KUKA KRL program: ps_p13060r5_all_resp_x1.src, ps_p13060r5_all_resp_x1.dat

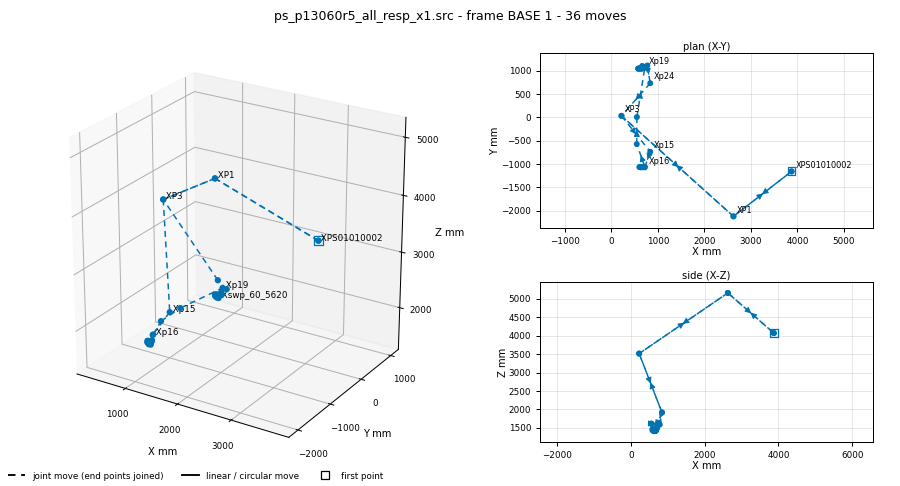
[picture p0: tool path of ps_p13060r5_all_resp_x1.src in frame BASE 1, 36 of 36 moves have a stored position in this frame; points joined in program order, loops and branches not executed]
--- ps_p13060r5_all_resp_x1.src ---
&ACCESS RVO1
&REL 27
&COMMENT SOLDA ACTROS GUN X1
&PARAM DISKPATH = KRC:\R1\Program
DEF ps_p13060r5_all_resp_x1( )
;FOLD INI
  ;FOLD BASISTECH INI
    GLOBAL INTERRUPT DECL 3 WHEN $STOPMESS==TRUE DO IR_STOPM ( )
    INTERRUPT ON 3
    BAS (#INITMOV,0 )
  ;ENDFOLD (BASISTECH INI)
;FOLD SPOTTECH INI
USERSPOT(#INIT)
;ENDFOLD (SPOTTECH INI)
;FOLD GRIPPERTECH INI

;ENDFOLD (GRIPPERTECH INI)
  ;FOLD USER INI
    ;Make your modifications here

     ;FOLD COLLISION_V_3.01 INI ;%{E}
        IF (COLLISION_DATA[1].I_NR>0) THEN
          GLOBAL INTERRUPT DECL 21 WHEN $IN[COLLISION_DATA[1].I_NR]==FALSE DO COLLSTOP (1,0 )
        ENDIF
        IF (COLLISION_DATA[2].I_NR>0) THEN
          GLOBAL INTERRUPT DECL 22 WHEN $IN[COLLISION_DATA[2].I_NR]==FALSE DO COLLSTOP (2,0 )
        ENDIF
        IF (COLLISION_DATA[3].I_NR>0) THEN
          GLOBAL INTERRUPT DECL 23 WHEN $IN[COLLISION_DATA[3].I_NR]==FALSE DO COLLSTOP (3,0 )
        ENDIF
        IF (COLLISION_DATA[4].I_NR>0) THEN
          GLOBAL INTERRUPT DECL 24 WHEN $IN[COLLISION_DATA[4].I_NR]==FALSE DO COLLSTOP (4,0 )
        ENDIF
     ;ENDFOLD (Collision)

  ;ENDFOLD (USER INI)
;ENDFOLD (INI)

; Caracterização dos meios de produção: P13.060-R5
; Versão atual: 17/07/2013 Nome: Solda Respot X1
; Change: LTA/LTA/MGS/MHSB/STB

chk_w1_wechs_ok ( )           ; VERIFICAÇÃO DE FERRAMENA: X1

;FOLD PTP PS01010002 Vel=100 % PDAT23 Tool[1]:Gun X1 Base[1]:Actros;%{PE}%R 8.2.20,%MKUKATPBASIS,%CMOVE,%VPTP,%P 1:PTP, 2:PS01010002, 3:, 5:100, 7:PDAT23
$BWDSTART=FALSE
PDAT_ACT=PPDAT23
FDAT_ACT=FPS01010002
BAS(#PTP_PARAMS,100)
PTP XPS01010002
;ENDFOLD

IF MaxStandMenge (3) THEN
 MaxStandmengeErreicht (3)
ENDIF

IF Elektrodenwechsel (3) THEN
 e_Fraes_1 ()
ENDIF


;FOLD PTP P1 CONT Vel=100 % PDAT15 Tool[1]:Gun X1 Base[1]:Actros;%{PE}%R 8.2.20,%MKUKATPBASIS,%CMOVE,%VPTP,%P 1:PTP, 2:P1, 3:C_DIS, 5:100, 7:PDAT15
$BWDSTART=FALSE
PDAT_ACT=PPDAT15
FDAT_ACT=FP1
BAS(#PTP_PARAMS,100)
PTP XP1 C_DIS
;ENDFOLD
;FOLD PTP P3 CONT Vel=100 % PDAT18 Tool[1]:Gun X1 Base[1]:Actros;%{PE}%R 8.2.20,%MKUKATPBASIS,%CMOVE,%VPTP,%P 1:PTP, 2:P3, 3:C_DIS, 5:100, 7:PDAT18
$BWDSTART=FALSE
PDAT_ACT=PPDAT18
FDAT_ACT=FP3
BAS(#PTP_PARAMS,100)
PTP XP3 C_DIS
;ENDFOLD
;FOLD PTP p15 CONT Vel=100 % P_OLP2 Tool[1]:Gun X1 Base[1]:Actros;%{PE}%R 8.2.20,%MKUKATPBASIS,%CMOVE,%VPTP,%P 1:PTP, 2:p15, 3:C_DIS, 5:100, 7:P_OLP2
$BWDSTART=FALSE
PDAT_ACT=PP_OLP2
FDAT_ACT=Fp15
BAS(#PTP_PARAMS,100)
PTP Xp15 C_DIS
;ENDFOLD

;FOLD Collision.Monitoring_1_On ;%{PE}%MKUKATPUSER
COLLSTOP( 1, 1 ) ;Interrupt-Controlled
;ENDFOLD

;FOLD OUT 3339 'R5 SOLDANDO' State=TRUE ;%{PE}%R 8.2.20,%MKUKATPBASIS,%COUT,%VOUTX,%P 2:3339, 3:R5 SOLDANDO, 5:TRUE, 6:
$OUT[3339]=TRUE
;ENDFOLD
;FOLD OUT 3340 'locking-signal PLC' State=FALSE ;%{PE}%R 8.2.20,%MKUKATPBASIS,%COUT,%VOUTX,%P 2:3340, 3:locking-signal PLC, 5:FALSE, 6:
$OUT[3340]=FALSE
;ENDFOLD

;FOLD PTP p16 CONT Vel=100 % P_OLP3 Tool[1]:Gun X1 Base[1]:Actros;%{PE}%R8.2,%MKUKATPBASIS,%CMOVE,%VPTP,%P 1:PTP, 2:p16, 3:C_DIS, 5:100, 7:P_OLP3
$BWDSTART = FALSE
PDAT_ACT= PP_OLP3
FDAT_ACT= Fp16
BAS(#PTP_PARAMS,100)
PTP Xp16 C_DIS
;ENDFOLD
;FOLD PTP P7 CONT Vel=100 % PDAT22 Tool[1]:Gun X1 Base[1]:Actros;%{PE}%R 8.2.20,%MKUKATPBASIS,%CMOVE,%VPTP,%P 1:PTP, 2:P7, 3:C_DIS, 5:100, 7:PDAT22
$BWDSTART=FALSE
PDAT_ACT=PPDAT22
FDAT_ACT=FP7
BAS(#PTP_PARAMS,100)
PTP XP7 C_DIS
;ENDFOLD
;FOLD PTP p17 PDAT1 RETR CLS Gun=3 Tool[1]:Gun X1 Base[1]:Actros;%{PE}%R 8.2.2,%MKUKATPSPOT,%CRETR,%VPTP,%P 1:PTP, 2:p17, 3:, 5:100, 7:PDAT1, 9:#CLO, 11:3, 13:#FIRST
$BWDSTART=FALSE
PDAT_ACT=PPDAT1
FDAT_ACT=Fp17
BAS(#PTP_PARAMS,PPDAT1.VEL)
S_ACT.GUN=3
S_ACT.PAIR=#FIRST
S_ACT.RETR=#CLO
S_READY=FALSE
PTP Xp17
USERSPOT(#RETR, S_ACT)
WAIT FOR S_READY
;ENDFOLD

;FOLD ; SWP_60_5617;%{PE}%R 8.2.20,%MKUKATPBASIS,%CCOMMENT,%VNORMAL,%P 2:SWP_60_5617
;ENDFOLD
;FOLD PTP swp_60_5617 PDAT2 SPOT Gun=3 RETR CLS PGNO1=121 ACTIVE=1 Tool[1]:Gun X1 Base[1]:Actros;%{PE}%R 8.2.2,%MKUKATPSPOT,%CSPOT,%VPTP,%P 1:PTP, 2:swp_60_5617, 3:, 5:100, 7:PDAT2, 10:3, 12:#FIRST, 14:#CLO, 16:171, 18:1, 20:0, 22:0, 24:1, 25:NORMAL
$BWDSTART=FALSE
PDAT_ACT=PPDAT2
FDAT_ACT=Fswp_60_5617
BAS(#PTP_PARAMS,PPDAT2.VEL)
S_ACT.GUN=3
S_ACT.PAIR=SDEFAULT.PAIR
S_ACT.RETR=#CLO
S_ACT.CLO_TM=1
S_ACT.PGNO1=121
S_ACT.PGNO2=SDEFAULT.PGNO2
S_ACT.PRESS1=SDEFAULT.PRESS1
S_ACT.PRESS2=SDEFAULT.PRESS2
S_READY=FALSE
PTP Xswp_60_5617
USERSPOT(#SPOT, S_ACT)
WAIT FOR S_READY
;ENDFOLD

;FOLD ; SWP_60_5619;%{PE}%R 8.2.20,%MKUKATPBASIS,%CCOMMENT,%VNORMAL,%P 2:SWP_60_5619
;ENDFOLD
;FOLD PTP swp_60_5619 PDAT3 SPOT Gun=3 RETR CLS PGNO1=122 ACTIVE=1 Tool[1]:Gun X1 Base[1]:Actros;%{PE}%R 8.2.2,%MKUKATPSPOT,%CSPOT,%VPTP,%P 1:PTP, 2:swp_60_5619, 3:, 5:100, 7:PDAT3, 10:3, 12:#FIRST, 14:#CLO, 16:172, 18:1, 20:0, 22:0, 24:1, 25:NORMAL
$BWDSTART=FALSE
PDAT_ACT=PPDAT3
FDAT_ACT=Fswp_60_5619
BAS(#PTP_PARAMS,PPDAT3.VEL)
S_ACT.GUN=3
S_ACT.PAIR=SDEFAULT.PAIR
S_ACT.RETR=#CLO
S_ACT.CLO_TM=1
S_ACT.PGNO1=122
S_ACT.PGNO2=SDEFAULT.PGNO2
S_ACT.PRESS1=SDEFAULT.PRESS1
S_ACT.PRESS2=SDEFAULT.PRESS2
S_READY=FALSE
PTP Xswp_60_5619
USERSPOT(#SPOT, S_ACT)
WAIT FOR S_READY
;ENDFOLD

;FOLD ; SWP_60_5615;%{PE}%R 8.2.20,%MKUKATPBASIS,%CCOMMENT,%VNORMAL,%P 2:SWP_60_5615
;ENDFOLD
;FOLD PTP swp_60_5615 PDAT4 SPOT Gun=3 RETR CLS PGNO1=123 ACTIVE=1 Tool[1]:Gun X1 Base[1]:Actros;%{PE}%R 8.2.2,%MKUKATPSPOT,%CSPOT,%VPTP,%P 1:PTP, 2:swp_60_5615, 3:, 5:100, 7:PDAT4, 10:3, 12:#FIRST, 14:#CLO, 16:173, 18:1, 20:0, 22:0, 24:1, 25:NORMAL
$BWDSTART=FALSE
PDAT_ACT=PPDAT4
FDAT_ACT=Fswp_60_5615
BAS(#PTP_PARAMS,PPDAT4.VEL)
S_ACT.GUN=3
S_ACT.PAIR=SDEFAULT.PAIR
S_ACT.RETR=#CLO
S_ACT.CLO_TM=1
S_ACT.PGNO1=123
S_ACT.PGNO2=SDEFAULT.PGNO2
S_ACT.PRESS1=SDEFAULT.PRESS1
S_ACT.PRESS2=SDEFAULT.PRESS2
S_READY=FALSE
PTP Xswp_60_5615
USERSPOT(#SPOT, S_ACT)
WAIT FOR S_READY
;ENDFOLD

;FOLD ; SWP_60_5613;%{PE}%R 8.2.20,%MKUKATPBASIS,%CCOMMENT,%VNORMAL,%P 2:SWP_60_5613
;ENDFOLD
;FOLD PTP swp_60_5613 PDAT5 SPOT Gun=3 RETR CLS PGNO1=124 ACTIVE=1 Tool[1]:Gun X1 Base[1]:Actros;%{PE}%R 8.2.2,%MKUKATPSPOT,%CSPOT,%VPTP,%P 1:PTP, 2:swp_60_5613, 3:, 5:100, 7:PDAT5, 10:3, 12:#FIRST, 14:#CLO, 16:174, 18:1, 20:0, 22:0, 24:1, 25:NORMAL
$BWDSTART=FALSE
PDAT_ACT=PPDAT5
FDAT_ACT=Fswp_60_5613
BAS(#PTP_PARAMS,PPDAT5.VEL)
S_ACT.GUN=3
S_ACT.PAIR=SDEFAULT.PAIR
S_ACT.RETR=#CLO
S_ACT.CLO_TM=1
S_ACT.PGNO1=124
S_ACT.PGNO2=SDEFAULT.PGNO2
S_ACT.PRESS1=SDEFAULT.PRESS1
S_ACT.PRESS2=SDEFAULT.PRESS2
S_READY=FALSE
PTP Xswp_60_5613
USERSPOT(#SPOT, S_ACT)
WAIT FOR S_READY
;ENDFOLD

;FOLD LIN P8 CONT Vel=1 m/s CPDAT3 Tool[1]:Gun X1 Base[1]:Actros;%{PE}%R 8.2.20,%MKUKATPBASIS,%CMOVE,%VLIN,%P 1:LIN, 2:P8, 3:C_DIS C_DIS, 5:1, 7:CPDAT3
$BWDSTART=FALSE
LDAT_ACT=LCPDAT3
FDAT_ACT=FP8
BAS(#CP_PARAMS,1)
LIN XP8 C_DIS C_DIS
;ENDFOLD

;FOLD ; SWP_60_5611;%{PE}%R 8.2.20,%MKUKATPBASIS,%CCOMMENT,%VNORMAL,%P 2:SWP_60_5611
;ENDFOLD
;FOLD PTP swp_60_5611 PDAT6 SPOT Gun=3 RETR CLS PGNO1=125 ACTIVE=1 Tool[1]:Gun X1 Base[1]:Actros;%{PE}%R 8.2.2,%MKUKATPSPOT,%CSPOT,%VPTP,%P 1:PTP, 2:swp_60_5611, 3:, 5:100, 7:PDAT6, 10:3, 12:#FIRST, 14:#CLO, 16:175, 18:1, 20:0, 22:0, 24:1, 25:NORMAL
$BWDSTART=FALSE
PDAT_ACT=PPDAT6
FDAT_ACT=Fswp_60_5611
BAS(#PTP_PARAMS,PPDAT6.VEL)
S_ACT.GUN=3
S_ACT.PAIR=SDEFAULT.PAIR
S_ACT.RETR=#CLO
S_ACT.CLO_TM=1
S_ACT.PGNO1=125
S_ACT.PGNO2=SDEFAULT.PGNO2
S_ACT.PRESS1=SDEFAULT.PRESS1
S_ACT.PRESS2=SDEFAULT.PRESS2
S_READY=FALSE
PTP Xswp_60_5611
USERSPOT(#SPOT, S_ACT)
WAIT FOR S_READY
;ENDFOLD

;FOLD ; SWP_60_5605;%{PE}%R 8.2.20,%MKUKATPBASIS,%CCOMMENT,%VNORMAL,%P 2:SWP_60_5605
;ENDFOLD
;FOLD LIN swp_60_5605 CPDAT1 SPOT Gun=3 RETR CLS PGNO1=126 ACTIVE=1 Tool[1]:Gun X1 Base[1]:Actros;%{PE}%R 8.2.2,%MKUKATPSPOT,%CSPOT,%VLIN,%P 1:LIN, 2:swp_60_5605, 3:, 5:2, 7:CPDAT1, 10:3, 12:#FIRST, 14:#CLO, 16:176, 18:1, 20:0, 22:0, 24:1, 25:NORMAL
$BWDSTART=FALSE
LDAT_ACT=LCPDAT1
FDAT_ACT=Fswp_60_5605
BAS(#CP_PARAMS,LCPDAT1.VEL)
S_ACT.GUN=3
S_ACT.PAIR=SDEFAULT.PAIR
S_ACT.RETR=#CLO
S_ACT.CLO_TM=1
S_ACT.PGNO1=126
S_ACT.PGNO2=SDEFAULT.PGNO2
S_ACT.PRESS1=SDEFAULT.PRESS1
S_ACT.PRESS2=SDEFAULT.PRESS2
S_READY=FALSE
LIN Xswp_60_5605
USERSPOT(#SPOT, S_ACT)
WAIT FOR S_READY
;ENDFOLD

;FOLD ; SWP_60_5607;%{PE}%R 8.2.20,%MKUKATPBASIS,%CCOMMENT,%VNORMAL,%P 2:SWP_60_5607
;ENDFOLD
;FOLD LIN swp_60_5607 CPDAT4 SPOT Gun=3 RETR CLS PGNO1=127 ACTIVE=1 Tool[1]:Gun X1 Base[1]:Actros;%{PE}%R 8.2.2,%MKUKATPSPOT,%CSPOT,%VLIN,%P 1:LIN, 2:swp_60_5607, 3:, 5:2, 7:CPDAT4, 10:3, 12:#FIRST, 14:#CLO, 16:177, 18:1, 20:0, 22:0, 24:1, 25:NORMAL
$BWDSTART=FALSE
LDAT_ACT=LCPDAT4
FDAT_ACT=Fswp_60_5607
BAS(#CP_PARAMS,LCPDAT4.VEL)
S_ACT.GUN=3
S_ACT.PAIR=SDEFAULT.PAIR
S_ACT.RETR=#CLO
S_ACT.CLO_TM=1
S_ACT.PGNO1=127
S_ACT.PGNO2=SDEFAULT.PGNO2
S_ACT.PRESS1=SDEFAULT.PRESS1
S_ACT.PRESS2=SDEFAULT.PRESS2
S_READY=FALSE
LIN Xswp_60_5607
USERSPOT(#SPOT, S_ACT)
WAIT FOR S_READY
;ENDFOLD

;FOLD ; SWP_60_5609;%{PE}%R 8.2.20,%MKUKATPBASIS,%CCOMMENT,%VNORMAL,%P 2:SWP_60_5609
;ENDFOLD
;FOLD PTP swp_60_5609 PDAT9 SPOT Gun=3 RETR OPN PGNO1=128 ACTIVE=1 Tool[1]:Gun X1 Base[1]:Actros;%{PE}%R 8.2.2,%MKUKATPSPOT,%CSPOT,%VPTP,%P 1:PTP, 2:swp_60_5609, 3:, 5:100, 7:PDAT9, 10:3, 12:#FIRST, 14:#OPN, 16:178, 18:1, 20:0, 22:0, 24:1, 25:NORMAL
$BWDSTART=FALSE
PDAT_ACT=PPDAT9
FDAT_ACT=Fswp_60_5609
BAS(#PTP_PARAMS,PPDAT9.VEL)
S_ACT.GUN=3
S_ACT.PAIR=SDEFAULT.PAIR
S_ACT.RETR=#OPN
S_ACT.CLO_TM=1
S_ACT.PGNO1=128
S_ACT.PGNO2=SDEFAULT.PGNO2
S_ACT.PRESS1=SDEFAULT.PRESS1
S_ACT.PRESS2=SDEFAULT.PRESS2
S_READY=FALSE
PTP Xswp_60_5609
USERSPOT(#SPOT, S_ACT)
WAIT FOR S_READY
;ENDFOLD

;FOLD PTP p18 CONT Vel=100 % P_OLP13 Tool[1]:Gun X1 Base[1]:Actros;%{PE}%R8.2,%MKUKATPBASIS,%CMOVE,%VPTP,%P 1:PTP, 2:p18, 3:C_DIS, 5:100, 7:P_OLP13
$BWDSTART = FALSE
PDAT_ACT= PP_OLP13
FDAT_ACT= Fp18
BAS(#PTP_PARAMS,100)
PTP Xp18 C_DIS
;ENDFOLD
;FOLD PTP P6 CONT Vel=100 % PDAT21 Tool[1]:Gun X1 Base[1]:Actros;%{PE}%R 8.2.20,%MKUKATPBASIS,%CMOVE,%VPTP,%P 1:PTP, 2:P6, 3:C_DIS, 5:100, 7:PDAT21
$BWDSTART=FALSE
PDAT_ACT=PPDAT21
FDAT_ACT=FP6
BAS(#PTP_PARAMS,100)
PTP XP6 C_DIS
;ENDFOLD

;FOLD Collision.Monitoring_1_Off . ;%{PE}%MKUKATPUSER
COLLSTOP( 1, 2+0 )
;ENDFOLD
;FOLD Collision.Monitoring_2_On ;%{PE}%MKUKATPUSER
COLLSTOP( 2, 1 ) ;Interrupt-Controlled
;ENDFOLD

;FOLD PTP p26 CONT Vel=100 % PDAT10 Tool[1]:Gun X1 Base[1]:Actros;%{PE}%R 8.2.20,%MKUKATPBASIS,%CMOVE,%VPTP,%P 1:PTP, 2:p26, 3:C_DIS, 5:100, 7:PDAT10
$BWDSTART=FALSE
PDAT_ACT=PPDAT10
FDAT_ACT=Fp26
BAS(#PTP_PARAMS,100)
PTP Xp26 C_DIS
;ENDFOLD
;FOLD PTP p19 CONT Vel=100 % P_OLP14 Tool[1]:Gun X1 Base[1]:Actros;%{PE}%R8.2,%MKUKATPBASIS,%CMOVE,%VPTP,%P 1:PTP, 2:p19, 3:C_DIS, 5:100, 7:P_OLP14
$BWDSTART = FALSE
PDAT_ACT= PP_OLP14
FDAT_ACT= Fp19
BAS(#PTP_PARAMS,100)
PTP Xp19 C_DIS
;ENDFOLD
;FOLD PTP p20 CONT Vel=100 % PDAT12 Tool[1]:Gun X1 Base[1]:Actros;%{PE}%R 8.2.20,%MKUKATPBASIS,%CMOVE,%VPTP,%P 1:PTP, 2:p20, 3:C_DIS, 5:100, 7:PDAT12
$BWDSTART=FALSE
PDAT_ACT=PPDAT12
FDAT_ACT=Fp20
BAS(#PTP_PARAMS,100)
PTP Xp20 C_DIS
;ENDFOLD

;FOLD ; SWP_60_5610;%{PE}%R 8.2.20,%MKUKATPBASIS,%CCOMMENT,%VNORMAL,%P 2:SWP_60_5610
;ENDFOLD
;FOLD PTP swp_60_5610 PDAT13 SPOT Gun=3 RETR CLS PGNO1=129 ACTIVE=1 Tool[1]:Gun X1 Base[1]:Actros;%{PE}%R 8.2.2,%MKUKATPSPOT,%CSPOT,%VPTP,%P 1:PTP, 2:swp_60_5610, 3:, 5:100, 7:PDAT13, 10:3, 12:#FIRST, 14:#CLO, 16:179, 18:1, 20:0, 22:0, 24:1, 25:NORMAL
$BWDSTART=FALSE
PDAT_ACT=PPDAT13
FDAT_ACT=Fswp_60_5610
BAS(#PTP_PARAMS,PPDAT13.VEL)
S_ACT.GUN=3
S_ACT.PAIR=SDEFAULT.PAIR
S_ACT.RETR=#CLO
S_ACT.CLO_TM=1
S_ACT.PGNO1=129
S_ACT.PGNO2=SDEFAULT.PGNO2
S_ACT.PRESS1=SDEFAULT.PRESS1
S_ACT.PRESS2=SDEFAULT.PRESS2
S_READY=FALSE
PTP Xswp_60_5610
USERSPOT(#SPOT, S_ACT)
WAIT FOR S_READY
;ENDFOLD

;FOLD ; SWP_60_5608;%{PE}%R 8.2.20,%MKUKATPBASIS,%CCOMMENT,%VNORMAL,%P 2:SWP_60_5608
;ENDFOLD
;FOLD PTP swp_60_5608 PDAT14 SPOT Gun=3 RETR CLS PGNO1=130 ACTIVE=1 Tool[1]:Gun X1 Base[1]:Actros;%{PE}%R 8.2.2,%MKUKATPSPOT,%CSPOT,%VPTP,%P 1:PTP, 2:swp_60_5608, 3:, 5:100, 7:PDAT14, 10:3, 12:#FIRST, 14:#CLO, 16:180, 18:1, 20:0, 22:0, 24:1, 25:NORMAL
$BWDSTART=FALSE
PDAT_ACT=PPDAT14
FDAT_ACT=Fswp_60_5608
BAS(#PTP_PARAMS,PPDAT14.VEL)
S_ACT.GUN=3
S_ACT.PAIR=SDEFAULT.PAIR
S_ACT.RETR=#CLO
S_ACT.CLO_TM=1
S_ACT.PGNO1=130
S_ACT.PGNO2=SDEFAULT.PGNO2
S_ACT.PRESS1=SDEFAULT.PRESS1
S_ACT.PRESS2=SDEFAULT.PRESS2
S_READY=FALSE
PTP Xswp_60_5608
USERSPOT(#SPOT, S_ACT)
WAIT FOR S_READY
;ENDFOLD

;FOLD ; SWP_60_5606;%{PE}%R8.2,%MKUKATPBASIS,%CCOMMENT,%VNORMAL,%P 2: SWP_60_5606
;ENDFOLD
;FOLD PTP swp_60_5606 P_OLP18 SPOT Gun=3 RETR CLS PGNO1=131 ACTIVE=1 Tool[1]:Gun X1 Base[1]:Actros;%{PE}%R 8.2.2,%MKUKATPSPOT,%CSPOT,%VPTP,%P 1:PTP, 2:swp_60_5606, 3:, 5:100, 7:P_OLP18, 10:3, 12:#FIRST, 14:#CLO, 16:181, 18:1, 20:1, 22:0, 24:1, 25:S_OLP11
$BWDSTART=FALSE
PDAT_ACT=PP_OLP18
FDAT_ACT=Fswp_60_5606
BAS(#PTP_PARAMS,PP_OLP18.VEL)
S_ACT.GUN=3
S_ACT.PAIR=SDEFAULT.PAIR
S_ACT.RETR=#CLO
S_ACT.CLO_TM=1
S_ACT.PGNO1=131
S_ACT.PGNO2=SDEFAULT.PGNO2
S_ACT.PRESS1=SDEFAULT.PRESS1
S_ACT.PRESS2=SDEFAULT.PRESS2
S_READY=FALSE
PTP Xswp_60_5606
USERSPOT(#SPOT, S_ACT)
WAIT FOR S_READY
;ENDFOLD

;FOLD ; SWP_60_5612;%{PE}%R8.2,%MKUKATPBASIS,%CCOMMENT,%VNORMAL,%P 2: SWP_60_5612
;ENDFOLD
;FOLD LIN swp_60_5612 CPDAT2 SPOT Gun=3 RETR CLS PGNO1=132 ACTIVE=1 Tool[1]:Gun X1 Base[1]:Actros;%{PE}%R 8.2.2,%MKUKATPSPOT,%CSPOT,%VLIN,%P 1:LIN, 2:swp_60_5612, 3:, 5:2, 7:CPDAT2, 10:3, 12:#FIRST, 14:#CLO, 16:182, 18:1, 20:1, 22:0, 24:1, 25:S_OLP12
$BWDSTART=FALSE
LDAT_ACT=LCPDAT2
FDAT_ACT=Fswp_60_5612
BAS(#CP_PARAMS,LCPDAT2.VEL)
S_ACT.GUN=3
S_ACT.PAIR=SDEFAULT.PAIR
S_ACT.RETR=#CLO
S_ACT.CLO_TM=1
S_ACT.PGNO1=132
S_ACT.PGNO2=SDEFAULT.PGNO2
S_ACT.PRESS1=SDEFAULT.PRESS1
S_ACT.PRESS2=SDEFAULT.PRESS2
S_READY=FALSE
LIN Xswp_60_5612
USERSPOT(#SPOT, S_ACT)
WAIT FOR S_READY
;ENDFOLD

;FOLD ; SWP_60_5614;%{PE}%R8.2,%MKUKATPBASIS,%CCOMMENT,%VNORMAL,%P 2: SWP_60_5614
;ENDFOLD
;FOLD PTP swp_60_5614 P_OLP20 SPOT Gun=3 RETR CLS PGNO1=133 ACTIVE=1 Tool[1]:Gun X1 Base[1]:Actros;%{PE}%R 8.2.2,%MKUKATPSPOT,%CSPOT,%VPTP,%P 1:PTP, 2:swp_60_5614, 3:, 5:100, 7:P_OLP20, 10:3, 12:#FIRST, 14:#CLO, 16:183, 18:1, 20:1, 22:0, 24:1, 25:S_OLP13
$BWDSTART=FALSE
PDAT_ACT=PP_OLP20
FDAT_ACT=Fswp_60_5614
BAS(#PTP_PARAMS,PP_OLP20.VEL)
S_ACT.GUN=3
S_ACT.PAIR=SDEFAULT.PAIR
S_ACT.RETR=#CLO
S_ACT.CLO_TM=1
S_ACT.PGNO1=133
S_ACT.PGNO2=SDEFAULT.PGNO2
S_ACT.PRESS1=SDEFAULT.PRESS1
S_ACT.PRESS2=SDEFAULT.PRESS2
S_READY=FALSE
PTP Xswp_60_5614
USERSPOT(#SPOT, S_ACT)
WAIT FOR S_READY
;ENDFOLD

;FOLD ; SWP_60_5616;%{PE}%R8.2,%MKUKATPBASIS,%CCOMMENT,%VNORMAL,%P 2: SWP_60_5616
;ENDFOLD
;FOLD PTP swp_60_5616 P_OLP21 SPOT Gun=3 RETR CLS PGNO1=134 ACTIVE=1 Tool[1]:Gun X1 Base[1]:Actros;%{PE}%R 8.2.2,%MKUKATPSPOT,%CSPOT,%VPTP,%P 1:PTP, 2:swp_60_5616, 3:, 5:100, 7:P_OLP21, 10:3, 12:#FIRST, 14:#CLO, 16:184, 18:1, 20:1, 22:0, 24:1, 25:S_OLP14
$BWDSTART=FALSE
PDAT_ACT=PP_OLP21
FDAT_ACT=Fswp_60_5616
BAS(#PTP_PARAMS,PP_OLP21.VEL)
S_ACT.GUN=3
S_ACT.PAIR=SDEFAULT.PAIR
S_ACT.RETR=#CLO
S_ACT.CLO_TM=1
S_ACT.PGNO1=134
S_ACT.PGNO2=SDEFAULT.PGNO2
S_ACT.PRESS1=SDEFAULT.PRESS1
S_ACT.PRESS2=SDEFAULT.PRESS2
S_READY=FALSE
PTP Xswp_60_5616
USERSPOT(#SPOT, S_ACT)
WAIT FOR S_READY
;ENDFOLD

;FOLD ; SWP_60_5620;%{PE}%R8.2,%MKUKATPBASIS,%CCOMMENT,%VNORMAL,%P 2: SWP_60_5620
;ENDFOLD
;FOLD PTP swp_60_5620 P_OLP22 SPOT Gun=3 RETR CLS PGNO1=135 ACTIVE=1 Tool[1]:Gun X1 Base[1]:Actros;%{PE}%R 8.2.2,%MKUKATPSPOT,%CSPOT,%VPTP,%P 1:PTP, 2:swp_60_5620, 3:, 5:100, 7:P_OLP22, 10:3, 12:#FIRST, 14:#CLO, 16:185, 18:1, 20:1, 22:0, 24:1, 25:S_OLP15
$BWDSTART=FALSE
PDAT_ACT=PP_OLP22
FDAT_ACT=Fswp_60_5620
BAS(#PTP_PARAMS,PP_OLP22.VEL)
S_ACT.GUN=3
S_ACT.PAIR=SDEFAULT.PAIR
S_ACT.RETR=#CLO
S_ACT.CLO_TM=1
S_ACT.PGNO1=135
S_ACT.PGNO2=SDEFAULT.PGNO2
S_ACT.PRESS1=SDEFAULT.PRESS1
S_ACT.PRESS2=SDEFAULT.PRESS2
S_READY=FALSE
PTP Xswp_60_5620
USERSPOT(#SPOT, S_ACT)
WAIT FOR S_READY
;ENDFOLD

;FOLD ; SWP_60_5618;%{PE}%R8.2,%MKUKATPBASIS,%CCOMMENT,%VNORMAL,%P 2: SWP_60_5618
;ENDFOLD
;FOLD LIN swp_60_5618 CPDAT5 SPOT Gun=3 RETR CLS PGNO1=136 ACTIVE=1 Tool[1]:Gun X1 Base[1]:Actros;%{PE}%R 8.2.2,%MKUKATPSPOT,%CSPOT,%VLIN,%P 1:LIN, 2:swp_60_5618, 3:, 5:2, 7:CPDAT5, 10:3, 12:#FIRST, 14:#CLO, 16:186, 18:1, 20:1, 22:0, 24:1, 25:S_OLP16
$BWDSTART=FALSE
LDAT_ACT=LCPDAT5
FDAT_ACT=Fswp_60_5618
BAS(#CP_PARAMS,LCPDAT5.VEL)
S_ACT.GUN=3
S_ACT.PAIR=SDEFAULT.PAIR
S_ACT.RETR=#CLO
S_ACT.CLO_TM=1
S_ACT.PGNO1=136
S_ACT.PGNO2=SDEFAULT.PGNO2
S_ACT.PRESS1=SDEFAULT.PRESS1
S_ACT.PRESS2=SDEFAULT.PRESS2
S_READY=FALSE
LIN Xswp_60_5618
USERSPOT(#SPOT, S_ACT)
WAIT FOR S_READY
;ENDFOLD

;FOLD PTP p21 P_OLP24 RETR OPN Gun=3 Tool[1]:Gun X1 Base[1]:Actros;%{PE}%R 8.2.2,%MKUKATPSPOT,%CRETR,%VPTP,%P 1:PTP, 2:p21, 3:, 5:100, 7:P_OLP24, 9:#OPN, 11:3, 13:#FIRST
$BWDSTART=FALSE
PDAT_ACT=PP_OLP24
FDAT_ACT=Fp21
BAS(#PTP_PARAMS,PP_OLP24.VEL)
S_ACT.GUN=3
S_ACT.PAIR=#FIRST
S_ACT.RETR=#OPN
S_READY=FALSE
PTP Xp21
USERSPOT(#RETR, S_ACT)
WAIT FOR S_READY
;ENDFOLD
;FOLD PTP p22 CONT Vel=100 % P_OLP25 Tool[1]:Gun X1 Base[1]:Actros;%{PE}%R 8.2.20,%MKUKATPBASIS,%CMOVE,%VPTP,%P 1:PTP, 2:p22, 3:C_DIS, 5:100, 7:P_OLP25
$BWDSTART=FALSE
PDAT_ACT=PP_OLP25
FDAT_ACT=Fp22
BAS(#PTP_PARAMS,100)
PTP Xp22 C_DIS
;ENDFOLD
;FOLD PTP p23 CONT Vel=100 % P_OLP26 Tool[1]:Gun X1 Base[1]:Actros;%{PE}%R8.2,%MKUKATPBASIS,%CMOVE,%VPTP,%P 1:PTP, 2:p23, 3:C_DIS, 5:100, 7:P_OLP26
$BWDSTART = FALSE
PDAT_ACT= PP_OLP26
FDAT_ACT= Fp23
BAS(#PTP_PARAMS,100)
PTP Xp23 C_DIS
;ENDFOLD

;FOLD OUT 3339 'R5 SOLDANDO' State=FALSE ;%{PE}%R 8.2.20,%MKUKATPBASIS,%COUT,%VOUTX,%P 2:3339, 3:R5 SOLDANDO, 5:FALSE, 6:
$OUT[3339]=FALSE
;ENDFOLD
;FOLD OUT 3340 'locking-signal PLC' State=TRUE ;%{PE}%R 8.2.20,%MKUKATPBASIS,%COUT,%VOUTX,%P 2:3340, 3:locking-signal PLC, 5:TRUE, 6:
$OUT[3340]=TRUE
;ENDFOLD

;FOLD PTP p24 CONT Vel=100 % P_OLP27 Tool[1]:Gun X1 Base[1]:Actros;%{PE}%R8.2,%MKUKATPBASIS,%CMOVE,%VPTP,%P 1:PTP, 2:p24, 3:C_DIS, 5:100, 7:P_OLP27
$BWDSTART = FALSE
PDAT_ACT= PP_OLP27
FDAT_ACT= Fp24
BAS(#PTP_PARAMS,100)
PTP Xp24 C_DIS
;ENDFOLD

;FOLD Collision.Monitoring_2_Off . ;%{PE}%MKUKATPUSER
COLLSTOP( 2, 2+0 )
;ENDFOLD
;FOLD PULSE 3334 'R5 SOLDA RESPOT ACTROS OK' State=TRUE Time=3 sec;%{PE}%R 8.2.20,%MKUKATPBASIS,%COUT,%VPULSE,%P 2:3334, 3:R5 SOLDA RESPOT ACTROS OK, 5:TRUE, 6:, 8:3
PULSE($OUT[3334], TRUE,3)
;ENDFOLD

;FOLD PTP P4 CONT Vel=100 % PDAT19 Tool[1]:Gun X1 Base[1]:Actros;%{PE}%R 8.2.20,%MKUKATPBASIS,%CMOVE,%VPTP,%P 1:PTP, 2:P4, 3:C_DIS, 5:100, 7:PDAT19
$BWDSTART=FALSE
PDAT_ACT=PPDAT19
FDAT_ACT=FP4
BAS(#PTP_PARAMS,100)
PTP XP4 C_DIS
;ENDFOLD
;FOLD PTP P5 CONT Vel=100 % PDAT20 Tool[1]:Gun X1 Base[1]:Actros;%{PE}%R 8.2.20,%MKUKATPBASIS,%CMOVE,%VPTP,%P 1:PTP, 2:P5, 3:C_DIS, 5:100, 7:PDAT20
$BWDSTART=FALSE
PDAT_ACT=PPDAT20
FDAT_ACT=FP5
BAS(#PTP_PARAMS,100)
PTP XP5 C_DIS
;ENDFOLD
;FOLD PTP P9 Vel=100 % PDAT24 Tool[1]:Gun X1 Base[1]:Actros;%{PE}%R 8.2.20,%MKUKATPBASIS,%CMOVE,%VPTP,%P 1:PTP, 2:P9, 3:, 5:100, 7:PDAT24
$BWDSTART=FALSE
PDAT_ACT=PPDAT24
FDAT_ACT=FP9
BAS(#PTP_PARAMS,100)
PTP XP9
;ENDFOLD


IF FraesAnf (3) THEN
 f_Fraes_1()
ENDIF

END

--- ps_p13060r5_all_resp_x1.dat ---
&ACCESS RVO1
&REL 27
&COMMENT SOLDA ACTROS GUN X1
&PARAM DISKPATH = KRC:\R1\Program
DEFDAT  ps_p13060r5_all_resp_x1
;FOLD EXTERNAL DECLARATIONS;%{PE}%MKUKATPBASIS,%CEXT,%VCOMMON,%P
;FOLD GRIPPERTECH EXT
EXT  H50 (INT  :IN,INT  :IN,INT  :IN,GRP_TYP  :IN )
;ENDFOLD (GRIPPERTECH EXT)
;FOLD SPOTTECH EXT
EXT  USERSPOT (S_COMMAND  :IN,SPOT_TYPE  :IN )
;ENDFOLD (SPOTTECH EXT)
;FOLD BASISTECH EXT;%{PE}%MKUKATPBASIS,%CEXT,%VEXT,%P
EXT  BAS (BAS_COMMAND  :IN,REAL  :IN )
DECL INT SUCCESS
;ENDFOLD (BASISTECH EXT)
;FOLD USER EXT;%{E}%MKUKATPUSER,%CEXT,%VEXT,%P
;Make your modifications here

;ENDFOLD (USER EXT)
;ENDFOLD (EXTERNAL DECLARATIONS)

;# ============ START PATH : swp_p13060r5_all_resp_x1 =============
DECL FDAT Fp15={TOOL_NO 1,BASE_NO 1,IPO_FRAME #BASE,POINT2[] " "}
DECL PDAT PP_OLP2={VEL 100.0,ACC 100.0,APO_DIST 100.0,APO_MODE #CDIS}
DECL E6POS Xp15={X 837.791992,Y -736.427002,Z 1918.34998,A -178.472504,B 55.2508011,C -112.721901,S 2,T 3}
DECL FDAT Fp16={TOOL_NO 1,BASE_NO 1,IPO_FRAME #BASE,POINT2[] " "}
DECL PDAT PP_OLP3={VEL 100.0,ACC 100.0,APO_DIST 100.0,APO_MODE #CDIS}
DECL E6POS Xp16={X 720.363708,Y -1071.90405,Z 1611.62195,A -179.997894,B 40.0071182,C -89.2487793,S 2,T 11,E1 0.0,E2 0.0,E3 0.0,E4 0.0,E5 0.0,E6 0.0}
DECL FDAT Fp17={TOOL_NO 1,BASE_NO 1,IPO_FRAME #BASE,POINT2[] " ",TQ_STATE FALSE}
DECL E6POS Xp17={X 694.566772,Y -1067.33704,Z 1480.99805,A 179.533905,B 40.5357018,C -89.6439514,S 2,T 11,E1 0.0,E2 0.0,E3 0.0,E4 0.0,E5 0.0,E6 0.0}
DECL FDAT Fswp_60_5617={TOOL_NO 1,BASE_NO 1,IPO_FRAME #BASE,POINT2[] " ",TQ_STATE FALSE}
DECL SPOT_TYPE SS_OLP1={GUN 1,PAIR #FIRST,RETR #CLO,CLO_TM 0,PGNO1 1,PRESS1 1.0,PGNO2 0,PRESS2 0.0}
DECL E6POS Xswp_60_5617={X 637.125427,Y -1069.78503,Z 1416.79797,A 179.512695,B 37.7575111,C -89.6578064,S 2,T 11,E1 0.0,E2 0.0,E3 0.0,E4 0.0,E5 0.0,E6 0.0}
DECL FDAT Fswp_60_5619={TOOL_NO 1,BASE_NO 1,IPO_FRAME #BASE,POINT2[] " ",TQ_STATE FALSE}
DECL SPOT_TYPE SS_OLP2={GUN 1,PAIR #FIRST,RETR #CLO,CLO_TM 0,PGNO1 1,PRESS1 1.0,PGNO2 0,PRESS2 0.0}
DECL E6POS Xswp_60_5619={X 674.626892,Y -1067.28101,Z 1419.23303,A -178.805893,B 40.6008301,C -88.5975037,S 2,T 11,E1 0.0,E2 0.0,E3 0.0,E4 0.0,E5 0.0,E6 0.0}
DECL FDAT Fswp_60_5615={TOOL_NO 1,BASE_NO 1,IPO_FRAME #BASE,POINT2[] " ",TQ_STATE FALSE}
DECL SPOT_TYPE SS_OLP3={GUN 1,PAIR #FIRST,RETR #CLO,CLO_TM 0,PGNO1 1,PRESS1 1.0,PGNO2 0,PRESS2 0.0}
DECL E6POS Xswp_60_5615={X 673.435181,Y -1067.70105,Z 1449.01001,A -178.806198,B 40.6008911,C -88.5973129,S 2,T 11,E1 0.0,E2 0.0,E3 0.0,E4 0.0,E5 0.0,E6 0.0}
DECL FDAT Fswp_60_5613={TOOL_NO 1,BASE_NO 1,IPO_FRAME #BASE,POINT2[] " "}
DECL SPOT_TYPE SS_OLP4={GUN 1,PAIR #FIRST,RETR #CLO,CLO_TM 0,PGNO1 1,PRESS1 1.0,PGNO2 0,PRESS2 0.0}
DECL E6POS Xswp_60_5613={X 637.172974,Y -1068.25098,Z 1446.42297,A -178.821198,B 39.5516205,C -88.6091309,S 2,T 11,E1 0.0,E2 0.0,E3 0.0,E4 0.0,E5 0.0,E6 0.0}
DECL FDAT Fswp_60_5611={TOOL_NO 1,BASE_NO 1,IPO_FRAME #BASE,POINT2[] " "}
DECL SPOT_TYPE SS_OLP5={GUN 1,PAIR #FIRST,RETR #CLO,CLO_TM 0,PGNO1 1,PRESS1 1.0,PGNO2 0,PRESS2 0.0}
DECL E6POS Xswp_60_5611={X 608.086914,Y -1067.16602,Z 1443.45801,A -179.012405,B 31.1713409,C -88.7301331,S 2,T 11,E1 0.0,E2 0.0,E3 0.0,E4 0.0,E5 0.0,E6 0.0}
DECL FDAT Fswp_60_5605={TOOL_NO 1,BASE_NO 1,IPO_FRAME #BASE,POINT2[] " "}
DECL SPOT_TYPE SS_OLP6={GUN 1,PAIR #FIRST,RETR #CLO,CLO_TM 0,PGNO1 1,PRESS1 1.0,PGNO2 0,PRESS2 0.0}
DECL E6POS Xswp_60_5605={X 609.177612,Y -1065.95801,Z 1471.69495,A -178.997696,B 15.2031298,C -88.7556763,S 2,T 11,E1 0.0,E2 0.0,E3 0.0,E4 0.0,E5 0.0,E6 0.0}
DECL FDAT Fswp_60_5607={TOOL_NO 1,BASE_NO 1,IPO_FRAME #BASE,POINT2[] " ",TQ_STATE FALSE}
DECL SPOT_TYPE SS_OLP7={GUN 1,PAIR #FIRST,RETR #CLO,CLO_TM 0,PGNO1 1,PRESS1 1.0,PGNO2 0,PRESS2 0.0}
DECL E6POS Xswp_60_5607={X 635.962524,Y -1066.53796,Z 1474.59595,A 177.543701,B 21.5745106,C -91.1538773,S 2,T 43,E1 0.0,E2 0.0,E3 0.0,E4 0.0,E5 0.0,E6 0.0}
DECL FDAT Fswp_60_5609={TOOL_NO 1,BASE_NO 1,IPO_FRAME #BASE,POINT2[] " "}
DECL SPOT_TYPE SS_OLP8={GUN 1,PAIR #FIRST,RETR #OPN,CLO_TM 0,PGNO1 1,PRESS1 1.0,PGNO2 0,PRESS2 0.0}
DECL E6POS Xswp_60_5609={X 672.785278,Y -1066.11096,Z 1477.26599,A 177.433807,B 26.6702309,C -91.4772797,S 2,T 43,E1 0.0,E2 0.0,E3 0.0,E4 0.0,E5 0.0,E6 0.0}
DECL FDAT Fp18={TOOL_NO 1,BASE_NO 1,IPO_FRAME #BASE,POINT2[] " "}
DECL PDAT PP_OLP13={VEL 100.0,ACC 100.0,APO_DIST 100.0,APO_MODE #CDIS}
DECL E6POS Xp18={X 720.190002,Y -1059.61304,Z 1611.57104,A 179.729996,B 20.0084991,C -89.3867035,S 2,T 11}
DECL FDAT Fp19={TOOL_NO 1,BASE_NO 1,IPO_FRAME #BASE,POINT2[] " "}
DECL PDAT PP_OLP14={VEL 100.0,ACC 100.0,APO_DIST 100.0,APO_MODE #CDIS}
DECL E6POS Xp19={X 720.442688,Y 1067.224,Z 1612.427,A -179.729797,B 20.0086594,C -90.6129532,S 2,T 2,E1 0.0,E2 0.0,E3 0.0,E4 0.0,E5 0.0,E6 0.0}
DECL FDAT Fp20={TOOL_NO 1,BASE_NO 1,IPO_FRAME #BASE,POINT2[] " ",TQ_STATE FALSE}
DECL E6POS Xp20={X 695.351379,Y 1082.38794,Z 1474.93005,A -179.573502,B 28.9461803,C -90.7650909,S 2,T 2,E1 0.0,E2 0.0,E3 0.0,E4 0.0,E5 0.0,E6 0.0}
DECL FDAT Fswp_60_5610={TOOL_NO 1,BASE_NO 1,IPO_FRAME #BASE,POINT2[] " "}
DECL SPOT_TYPE SS_OLP9={GUN 1,PAIR #FIRST,RETR #CLO,CLO_TM 0,PGNO1 1,PRESS1 1.0,PGNO2 0,PRESS2 0.0}
DECL E6POS Xswp_60_5610={X 651.329407,Y 1053.61401,Z 1470.08899,A -179.484207,B 32.148941,C -90.4953766,S 2,T 2,E1 0.0,E2 0.0,E3 0.0,E4 0.0,E5 0.0,E6 0.0}
DECL FDAT Fswp_60_5608={TOOL_NO 1,BASE_NO 1,IPO_FRAME #BASE,POINT2[] " "}
DECL SPOT_TYPE SS_OLP10={GUN 1,PAIR #FIRST,RETR #CLO,CLO_TM 0,PGNO1 1,PRESS1 1.0,PGNO2 0,PRESS2 0.0}
DECL E6POS Xswp_60_5608={X 608.985718,Y 1051.75806,Z 1470.50305,A -179.494598,B 21.9768505,C -90.4172592,S 2,T 2,E1 0.0,E2 0.0,E3 0.0,E4 0.0,E5 0.0,E6 0.0}
DECL FDAT Fswp_60_5606={TOOL_NO 1,BASE_NO 1,IPO_FRAME #BASE,POINT2[] " "}
DECL PDAT PP_OLP18={VEL 100.0,ACC 100.0,APO_DIST 0.0}
DECL SPOT_TYPE SS_OLP11={GUN 1,PAIR #FIRST,RETR #CLO,CLO_TM 0,PGNO1 1,PRESS1 1.0,PGNO2 0,PRESS2 0.0}
DECL E6POS Xswp_60_5606={X 578.524414,Y 1047.75098,Z 1463.854,A -179.497696,B 17.9471493,C -90.3690338,S 2,T 2,E1 0.0,E2 0.0,E3 0.0,E4 0.0,E5 0.0,E6 0.0}
DECL FDAT Fswp_60_5612={TOOL_NO 1,BASE_NO 1,IPO_FRAME #BASE,POINT2[] " "}
DECL SPOT_TYPE SS_OLP12={GUN 1,PAIR #FIRST,RETR #CLO,CLO_TM 0,PGNO1 1,PRESS1 1.0,PGNO2 0,PRESS2 0.0}
DECL E6POS Xswp_60_5612={X 580.710205,Y 1050.41699,Z 1432.87695,A -178.232193,B 26.2880497,C -89.5013504,S 2,T 2,E1 0.0,E2 0.0,E3 0.0,E4 0.0,E5 0.0,E6 0.0}
DECL FDAT Fswp_60_5614={TOOL_NO 1,BASE_NO 1,IPO_FRAME #BASE,POINT2[] " "}
DECL PDAT PP_OLP20={VEL 100.0,ACC 100.0,APO_DIST 0.0}
DECL SPOT_TYPE SS_OLP13={GUN 1,PAIR #FIRST,RETR #CLO,CLO_TM 0,PGNO1 1,PRESS1 1.0,PGNO2 0,PRESS2 0.0}
DECL E6POS Xswp_60_5614={X 611.156494,Y 1052.52405,Z 1436.51501,A -178.270294,B 28.0306892,C -89.6753387,S 2,T 2,E1 0.0,E2 0.0,E3 0.0,E4 0.0,E5 0.0,E6 0.0}
DECL FDAT Fswp_60_5616={TOOL_NO 1,BASE_NO 1,IPO_FRAME #BASE,POINT2[] " "}
DECL PDAT PP_OLP21={VEL 100.0,ACC 100.0,APO_DIST 0.0}
DECL SPOT_TYPE SS_OLP14={GUN 1,PAIR #FIRST,RETR #CLO,CLO_TM 0,PGNO1 1,PRESS1 1.0,PGNO2 0,PRESS2 0.0}
DECL E6POS Xswp_60_5616={X 649.708923,Y 1052.60596,Z 1436.89001,A -178.169098,B 28.2620296,C -89.4620972,S 2,T 2,E1 0.0,E2 0.0,E3 0.0,E4 0.0,E5 0.0,E6 0.0}
DECL FDAT Fswp_60_5620={TOOL_NO 1,BASE_NO 1,IPO_FRAME #BASE,POINT2[] " "}
DECL PDAT PP_OLP22={VEL 100.0,ACC 100.0,APO_DIST 0.0}
DECL SPOT_TYPE SS_OLP15={GUN 1,PAIR #FIRST,RETR #CLO,CLO_TM 0,PGNO1 1,PRESS1 1.0,PGNO2 0,PRESS2 0.0}
DECL E6POS Xswp_60_5620={X 648.585327,Y 1051.68201,Z 1410.70996,A -178.0746,B 34.4508705,C -89.3280106,S 2,T 2,E1 0.0,E2 0.0,E3 0.0,E4 0.0,E5 0.0,E6 0.0}
DECL FDAT Fswp_60_5618={TOOL_NO 1,BASE_NO 1,IPO_FRAME #BASE,POINT2[] " ",TQ_STATE FALSE}
DECL SPOT_TYPE SS_OLP16={GUN 1,PAIR #FIRST,RETR #CLO,CLO_TM 0,PGNO1 1,PRESS1 1.0,PGNO2 0,PRESS2 0.0}
DECL E6POS Xswp_60_5618={X 614.106323,Y 1053.00305,Z 1409.77002,A -178.013397,B 38.5371704,C -89.2914734,S 2,T 2,E1 0.0,E2 0.0,E3 0.0,E4 0.0,E5 0.0,E6 0.0}
DECL FDAT Fp21={TOOL_NO 1,BASE_NO 1,IPO_FRAME #BASE,POINT2[] " "}
DECL PDAT PP_OLP24={VEL 100.0,ACC 100.0,APO_DIST 100.0,APO_MODE #CDIS}
DECL E6POS Xp21={X 666.627686,Y 1058.40198,Z 1469.33105,A -178.781097,B 39.1957283,C -89.7718964,S 2,T 2,E1 0.0,E2 0.0,E3 0.0,E4 0.0,E5 0.0,E6 0.0}
DECL FDAT Fp22={TOOL_NO 1,BASE_NO 1,IPO_FRAME #BASE,POINT2[] " "}
DECL PDAT PP_OLP25={VEL 100.0,ACC 100.0,APO_DIST 100.0,APO_MODE #CDIS}
DECL E6POS Xp22={X 665.576782,Y 1106.58801,Z 1493.98303,A -178.776794,B 39.1956902,C -89.7690201,S 2,T 2,E1 0.0,E2 0.0,E3 0.0,E4 0.0,E5 0.0,E6 0.0}
DECL FDAT Fp23={TOOL_NO 1,BASE_NO 1,IPO_FRAME #BASE,POINT2[] " "}
DECL PDAT PP_OLP26={VEL 100.0,ACC 100.0,APO_DIST 100.0,APO_MODE #CDIS}
DECL E6POS Xp23={X 773.952026,Y 1115.85095,Z 1585.13599,A 178.0784,B 46.9954987,C -90.9132004,S 2,T 2}
DECL FDAT Fp24={TOOL_NO 1,BASE_NO 1,IPO_FRAME #BASE,POINT2[] " "}
DECL PDAT PP_OLP27={VEL 100.0,ACC 100.0,APO_DIST 100.0,APO_MODE #CDIS}
DECL E6POS Xp24={X 837.791992,Y 736.427002,Z 1918.34998,A 178.472504,B 55.2508011,C -67.2780991,S 2,T 10}
DECL SPOT_SUGG_T LAST_SPOT={GUN[] "1                       ",RETR_CMD[] "#CLO                    ",CHOISE[] "#FIRST                  ",CLO_TM[] "1                       ",PGNO1[] "1                       ",PRESS1[] "0                       ",PGNO2[] "1                       ",PRESS2[] "0                       ",SPOT_PARAMS[] "NORMAL                  "}
DECL PDAT PPDAT1={VEL 80.0,ACC 100.0,APO_DIST 100.0}
DECL PDAT PPDAT2={VEL 90.0,ACC 100.0,APO_DIST 100.0}
DECL PDAT PPDAT3={VEL 90.0,ACC 100.0,APO_DIST 100.0}
DECL PDAT PPDAT4={VEL 90.0,ACC 100.0,APO_DIST 100.0}
DECL PDAT PPDAT5={VEL 90.0,ACC 100.0,APO_DIST 100.0}
DECL PDAT PPDAT6={VEL 90.0,ACC 100.0,APO_DIST 100.0}
DECL PDAT PPDAT9={VEL 100.0,ACC 100.0,APO_DIST 100.0}
DECL E6POS XP26={X 550.643188,Y 8.66149235,Z 1617.41797,A 179.826004,B 18.7652893,C -90.2307587,S 2,T 11,E1 0.0,E2 0.0,E3 0.0,E4 0.0,E5 0.0,E6 0.0}
DECL FDAT Fp26={TOOL_NO 1,BASE_NO 1,IPO_FRAME #BASE,POINT2[] " ",TQ_STATE FALSE}
DECL PDAT PPDAT10={VEL 100.0,ACC 100.0,APO_DIST 100.0,APO_MODE #CDIS}
DECL PDAT PPDAT12={VEL 100.0,ACC 100.0,APO_DIST 100.0,APO_MODE #CDIS}
DECL PDAT PPDAT13={VEL 100.0,ACC 100.0,APO_DIST 100.0}
DECL PDAT PPDAT14={VEL 100.0,ACC 100.0,APO_DIST 100.0}
DECL LDAT LCPDAT1={VEL 2.0,ACC 100.0,APO_DIST 100.0,APO_FAC 50.0,AXIS_VEL 100.0,AXIS_ACC 100.0,ORI_TYP #VAR,CIRC_TYP #BASE,JERK_FAC 50.0,GEAR_JERK 50.0,EXAX_IGN 0}
DECL LDAT LCPDAT2={VEL 2.0,ACC 100.0,APO_DIST 100.0,APO_FAC 50.0,AXIS_VEL 100.0,AXIS_ACC 100.0,ORI_TYP #VAR,CIRC_TYP #BASE,JERK_FAC 50.0,GEAR_JERK 50.0,EXAX_IGN 0}
DECL E6POS XP1={X 2625.59204,Y -2124.58691,Z 5161.79199,A -86.5009079,B -77.870697,C -89.1861496,S 2,T 11,E1 0.0,E2 0.0,E3 0.0,E4 0.0,E5 0.0,E6 0.0}
DECL FDAT FP1={TOOL_NO 1,BASE_NO 1,IPO_FRAME #BASE,POINT2[] " ",TQ_STATE FALSE}
DECL PDAT PPDAT15={VEL 100.0,ACC 100.0,APO_DIST 100.0,APO_MODE #CDIS}
DECL PDAT PPDAT18={VEL 100.0,ACC 100.0,APO_DIST 100.0,APO_MODE #CDIS}
DECL E6POS XP3={X 219.480896,Y 35.14151,Z 3516.46509,A -179.212204,B -4.39048815,C -89.7597809,S 2,T 3,E1 0.0,E2 0.0,E3 0.0,E4 0.0,E5 0.0,E6 0.0}
DECL FDAT FP3={TOOL_NO 1,BASE_NO 1,IPO_FRAME #BASE,POINT2[] " ",TQ_STATE FALSE}
DECL PDAT PPDAT19={VEL 100.0,ACC 100.0,APO_DIST 100.0,APO_MODE #CDIS}
DECL E6POS XP4={X 219.485901,Y 35.1248703,Z 3516.48999,A -179.212006,B -4.39138222,C -89.7597427,S 2,T 3,E1 0.0,E2 0.0,E3 0.0,E4 0.0,E5 0.0,E6 0.0}
DECL FDAT FP4={TOOL_NO 1,BASE_NO 1,IPO_FRAME #BASE,POINT2[] " ",TQ_STATE FALSE}
DECL PDAT PPDAT20={VEL 100.0,ACC 100.0,APO_DIST 100.0,APO_MODE #CDIS}
DECL E6POS XP5={X 2625.58789,Y -2124.58105,Z 5161.7959,A -86.5011978,B -77.8708878,C -89.1859589,S 2,T 11,E1 0.0,E2 0.0,E3 0.0,E4 0.0,E5 0.0,E6 0.0}
DECL FDAT FP5={TOOL_NO 1,BASE_NO 1,IPO_FRAME #BASE,POINT2[] " ",TQ_STATE FALSE}
DECL E6POS XP6={X 548.382874,Y -571.695129,Z 1611.77905,A 179.270004,B 18.8461399,C -90.9016876,S 2,T 11,E1 0.0,E2 0.0,E3 0.0,E4 0.0,E5 0.0,E6 0.0}
DECL FDAT FP6={TOOL_NO 1,BASE_NO 1,IPO_FRAME #BASE,POINT2[] " ",TQ_STATE FALSE}
DECL PDAT PPDAT21={VEL 100.0,ACC 100.0,APO_DIST 100.0,APO_MODE #CDIS}
DECL E6POS XP7={X 698.267273,Y -1063.01294,Z 1504.32898,A 179.617798,B 40.4430504,C -89.5728836,S 2,T 11,E1 0.0,E2 0.0,E3 0.0,E4 0.0,E5 0.0,E6 0.0}
DECL FDAT FP7={TOOL_NO 1,BASE_NO 1,IPO_FRAME #BASE,POINT2[] " ",TQ_STATE FALSE}
DECL PDAT PPDAT22={VEL 100.0,ACC 100.0,APO_DIST 5.0,APO_MODE #CDIS}
DECL E6POS XP8={X 616.294312,Y -1065.22803,Z 1442.66797,A -178.994003,B 33.5643005,C -88.6861572,S 2,T 11,E1 0.0,E2 0.0,E3 0.0,E4 0.0,E5 0.0,E6 0.0}
DECL FDAT FP8={TOOL_NO 1,BASE_NO 1,IPO_FRAME #BASE,POINT2[] " ",TQ_STATE FALSE}
DECL LDAT LCPDAT3={VEL 2.0,ACC 100.0,APO_DIST 2.0,APO_FAC 50.0,AXIS_VEL 100.0,AXIS_ACC 100.0,ORI_TYP #VAR,CIRC_TYP #BASE,JERK_FAC 50.0,GEAR_JERK 50.0,EXAX_IGN 0}
DECL LDAT LCPDAT4={VEL 1.0,ACC 100.0,APO_DIST 100.0,APO_FAC 50.0,AXIS_VEL 100.0,AXIS_ACC 100.0,ORI_TYP #VAR,CIRC_TYP #BASE,JERK_FAC 50.0,GEAR_JERK 50.0,EXAX_IGN 0}
DECL LDAT LCPDAT5={VEL 1.0,ACC 100.0,APO_DIST 100.0,APO_FAC 50.0,AXIS_VEL 100.0,AXIS_ACC 100.0,ORI_TYP #VAR,CIRC_TYP #BASE,JERK_FAC 50.0,GEAR_JERK 50.0,EXAX_IGN 0}
DECL E6POS XPS01010002={X 3873.65698,Y -1159.58105,Z 4073.08301,A 18.1216106,B -0.0244571492,C -112.231796,S 2,T 3,E1 0.0,E2 0.0,E3 0.0,E4 0.0,E5 0.0,E6 0.0}
DECL FDAT FPS01010002={TOOL_NO 1,BASE_NO 1,IPO_FRAME #BASE,POINT2[] " ",TQ_STATE FALSE}
DECL PDAT PPDAT23={VEL 100.0,ACC 100.0,APO_DIST 5.0,APO_MODE #CDIS}
DECL E6POS XP9={X 3873.65503,Y -1159.58398,Z 4073.08594,A 18.1212502,B -0.0245757699,C -112.231903,S 2,T 3,E1 0.0,E2 0.0,E3 0.0,E4 0.0,E5 0.0,E6 0.0}
DECL FDAT FP9={TOOL_NO 1,BASE_NO 1,IPO_FRAME #BASE,POINT2[] " ",TQ_STATE FALSE}
DECL PDAT PPDAT24={VEL 100.0,ACC 100.0,APO_DIST 5.0,APO_MODE #CDIS}
ENDDAT
